{attribute 'no_explicit_call' := 'Do not call the body - Stick to OOP'}
(* XPlanar Environment - 1 per associated XPlanar 
	The Planar environment is a software object that represents the two-dimensional XPlanar stator surface. Together with Planar movers in a group, 
	it prevents collisions of the movers with the edge of the surface. *)
FUNCTION_BLOCK FB_XP_Environment EXTENDS FB_CH_Object IMPLEMENTS I_XP_Environment
VAR
	//Link to Planar-Environment object
	fbEnvironment : MC_PlanarEnvironment;
	fbUtilityEnvirement : FB_TcIoXPlanarEnvironment;
	
	{attribute 'hide'}  
	bInitDone :BOOL := FALSE;
	{attribute 'hide'}
	ipXpSystem : I_XP_System_Registration;
	{attribute 'hide'}               	
	fbFeedback 			: FB_XP_Feedback(ipSourceInfo := fbSourceInfo);	
	{attribute 'hide'}                   	
	eActiveCommand 		: CHALET_Nc.E_NcAxisCommands := CHALET_Nc.E_NcAxisCommands.None;
	{attribute 'hide'}
	bCollisionCheckEnabled : BOOL := TRUE;
	{attribute 'hide'}
	fMoverOffsetWarning : LREAL := 2.0; //[mm]
	{attribute 'hide'}
	fMoverOffsetError: LREAL := 0.0;//[mm]
	{attribute 'hide'}
	eMoverDetectionStatus : MoverDetectionStatus;
	{attribute 'hide'}
	eMoverDetectionStatusLastCycle : MoverDetectionStatus;
END_VAR


// Planar-Feedback objects
VAR
	{attribute 'hide'} 
	fbFeedbackAddToGrp : MC_PlanarFeedback;
	{attribute 'hide'} 
	fbFeedbackRmvFromGrp : MC_PlanarFeedback;
	{attribute 'hide'} 
	fbFeedbackConfigure : MC_PlanarFeedback;
	{attribute 'hide'} 
	fbFeedbackClear : MC_PlanarFeedback;
END_VAR

METHOD AddToGroup : HRESULT
VAR_INPUT
	iGroup : I_XP_Group;
END_VAR
IF NOT THIS^.fbFeedback.Busy THEN
	THIS^.eActiveCommand 				:= CHALET_NC.E_NcAxisCommands.AddToGroupe;
	THIS^.fbFeedback.ActiveCommand 		:= TO_STRING(THIS^.eActiveCommand);	
	THIS^.fbFeedback.LastCommandAccepted:= TRUE;		
	THIS^.fbFeedback.Busy 				:= TRUE;
	
	iGroup.AddEnvironment(THIS^.fbEnvironment, THIS^.fbFeedbackAddToGrp);
	AddToGroup := S_OK;
ELSE
	AddToGroup := S_FALSE;
	THIS^.fbFeedback.LastCommandAccepted:= FALSE;	
END_IF
END_METHOD

(* Clears the Planar Environment (stators and boundary). *)
METHOD Clear : HRESULT
THIS^.eActiveCommand 				:= CHALET_NC.E_NcAxisCommands.Clear;
THIS^.fbFeedback.ActiveCommand 		:= TO_STRING(THIS^.eActiveCommand);	
THIS^.fbFeedback.LastCommandAccepted:= TRUE;		
THIS^.fbFeedback.Busy 				:= TRUE;

THIS^.fbEnvironment.Clear(commandFeedback:=THIS^.fbFeedbackClear);
Clear := S_OK;
END_METHOD

{attribute 'monitoring':='call'}
(* If Enable, the movers are checked for collisions with each other.
Warning and error can have their own size offsets.
The error leads to a stop with higher dynamics.
In simulation, an error does not lead to a stop *)
PROPERTY CollisionCheck : BOOL
GET
CollisionCheck := THIS^.bCollisionCheckEnabled;
END_GET
SET
THIS^.bCollisionCheckEnabled := CollisionCheck;
END_SET
END_PROPERTY

//Return an interface to the mover if a collision is active else return 0. The check stops after the first collision found
METHOD PROTECTED CollisionDetectionAlgorithm : I_XP_Mover
VAR_INPUT
	ipListOfMovers : I_CH_LIST;
	fOffsetMoverSize : LREAL := 1.0; //Offset on the mover dimension from the MC3 mover object [mm];
END_VAR
VAR
	aPointsMover1 : ARRAY[0..3] OF  Tc3_Physics.PositionXY;
	aPointsEachMover : ARRAY[0..3] OF  Tc3_Physics.PositionXY;
	aPointsDelta : ARRAY[0..3] OF  Tc3_Physics.PositionXY;
	
	fMoverWidth, fMoverHight : LREAL;
	fMoverXPos, fMoverYPos, fMoverCPos : LREAL;
	
	ipMover1, ipEachMover : I_XP_Mover;
	fbListOfMoverToCheck : FB_CH_List;
	
	fAngle : LREAL;
	a, b, c: LREAL;
	Pa, Pb, Pc : REFERENCE TO Tc3_Physics.PositionXY;
	fcos : LREAL;
	
	nIdx, nIdxMover1, nIdxPlus1 : UINT;
	ipMover2CollisionFound : I_XP_Mover;
END_VAR
//Get all mover in a list
fbListOfMoverToCheck.Duplicate(ipListOfMovers);



//Check list for invalide Act Pos - ex.: if mover is not found 
fbListOfMoverToCheck.ResetIterator();
WHILE fbListOfMoverToCheck.HasNextObject() DO
	__QUERYINTERFACE(fbListOfMoverToCheck.GetNextObject(),ipMover1);
	
	IF ipMover1.MoverIsNotPresent THEN 		
		//remove from list
		fbListOfMoverToCheck.RemoveObject(ipMover1);
		
	END_IF
END_WHILE



fbListOfMoverToCheck.ResetIterator();
WHILE fbListOfMoverToCheck.HasNextObject() DO
	//get first mover in list,
	__QUERYINTERFACE(fbListOfMoverToCheck.GetNextObject(),ipMover1);
	
	fMoverXPos := ipMover1.PositionAct.x;
	fMoverYPos := ipMover1.PositionAct.y;
	fMoverCPos := ipMover1.PositionAct.c;
		
	//Get corner points of the rectangle 
	fMoverWidth := ipMover1.MoverWidth - fOffsetMoverSize;
	fMoverHight := ipMover1.MoverHeight - fOffsetMoverSize;
	aPointsMover1[0].SetValuesXY(x:= -fMoverWidth/2, y:= -fMoverHight/2);//Bottom Left
	aPointsMover1[1].SetValuesXY(x:= -fMoverWidth/2, y:=  fMoverHight/2);//Top Left
	aPointsMover1[2].SetValuesXY(x:=  fMoverWidth/2, y:=  fMoverHight/2);//Top Ritgh
	aPointsMover1[3].SetValuesXY(x:=  fMoverWidth/2, y:= -fMoverHight/2);//Bottom Rigth
	
	//Rotation of the mover
	F_RotatePositionXY(aPointsMover1[0], fMoverCPos);
	F_RotatePositionXY(aPointsMover1[1], fMoverCPos);
	F_RotatePositionXY(aPointsMover1[2], fMoverCPos);
	F_RotatePositionXY(aPointsMover1[3], fMoverCPos);
	
	//shift to mover coordinates
	aPointsMover1[0].ShiftByXY(dx:= fMoverXPos, dy:= fMoverYPos);
	aPointsMover1[1].ShiftByXY(dx:= fMoverXPos, dy:= fMoverYPos);
	aPointsMover1[2].ShiftByXY(dx:= fMoverXPos, dy:= fMoverYPos);
	aPointsMover1[3].ShiftByXY(dx:= fMoverXPos, dy:= fMoverYPos);
	
	
	//do an check for all mover
	fbListOfMoverToCheck.ResetIterator();
	WHILE fbListOfMoverToCheck.HasNextObject() DO
		__QUERYINTERFACE(fbListOfMoverToCheck.GetNextObject(),ipEachMover);
		
		//Skip if same
		IF ipEachMover = ipMover1 THEN
			CONTINUE;
		END_IF
		
		//Skip if far away
		IF (MAX(ipEachMover.MoverHeight, ipEachMover.MoverWidth) + MAX(ipMover1.MoverHeight, ipMover1.MoverWidth) + fOffsetMoverSize) < F_DistXYVectors(ipEachMover.PositionAct, ipMover1.PositionAct) THEN
			CONTINUE;
		END_IF
		
		
		fMoverXPos := ipEachMover.PositionAct.x;
		fMoverYPos := ipEachMover.PositionAct.y;
		fMovercPos := ipEachMover.PositionAct.c;
		
		//Get corner points of the rectangle 
		fMoverWidth := ipEachMover.MoverWidth - fOffsetMoverSize;
		fMoverHight := ipEachMover.MoverHeight - fOffsetMoverSize;
		aPointsEachMover[0].SetValuesXY(x:= -fMoverWidth/2, y:= -fMoverHight/2);//Bottom Left
		aPointsEachMover[1].SetValuesXY(x:= -fMoverWidth/2, y:=  fMoverHight/2);//Top Left
		aPointsEachMover[2].SetValuesXY(x:=  fMoverWidth/2, y:=  fMoverHight/2);//Top Ritgh
		aPointsEachMover[3].SetValuesXY(x:=  fMoverWidth/2, y:= -fMoverHight/2);//Bottom Rigth

		//Rotation of the mover
		F_RotatePositionXY(aPointsEachMover[0], fMoverCPos);
		F_RotatePositionXY(aPointsEachMover[1], fMoverCPos);
		F_RotatePositionXY(aPointsEachMover[2], fMoverCPos);
		F_RotatePositionXY(aPointsEachMover[3], fMoverCPos);
		
		//shift to mover coordinates
		aPointsEachMover[0].ShiftByXY(dx:= fMoverXPos, dy:= fMoverYPos);
		aPointsEachMover[1].ShiftByXY(dx:= fMoverXPos, dy:= fMoverYPos);
		aPointsEachMover[2].ShiftByXY(dx:= fMoverXPos, dy:= fMoverYPos);
		aPointsEachMover[3].ShiftByXY(dx:= fMoverXPos, dy:= fMoverYPos);		
		
		//check each corener if inside each mover
		FOR nIdxMover1 := 0 TO 3 DO
			
			(* A triangle is created between a corner point of Mover1 (point a) and two corner points of Mover2 (points B and C). 
			All corner points of Mover2 are now tested one after the other. If the sum of all angles "a" is 360 degrees, 
			then point A is inside mover 2 and there is a collision *)
			fAngle := 0;
			FOR nIdx := 0 TO 3 DO
				nIdxPlus1 := ((nIdx+1)MOD 4);
			
				Pa REF= aPointsMover1[nIdxMover1];
				Pb REF= aPointsEachMover[nIdx];
				Pc REF= aPointsEachMover[nIdxPlus1];					
				

				a := SQRT(EXPT((Pb.x - Pc.x),2)+EXPT((Pb.y - Pc.y),2));
				b := SQRT(EXPT((Pa.x - Pc.x),2)+EXPT((Pa.y - Pc.y),2));
				c := SQRT(EXPT((Pa.x - Pb.x),2)+EXPT((Pa.y - Pb.y),2));
				
				
				IF b=0 OR c=0 THEN
					//Error - Return the found mover
					CollisionDetectionAlgorithm := ipMover1;
					//with which mover is the collision
					ipMover2CollisionFound := ipEachMover;
					RETURN;
				ELSE
					(*  a/sin(α) = b/sin(β) = c/sin(γ) *)
					fcos := (EXPT(b,2) + EXPT(c,2) - EXPT(a,2))/(2*b*c);
					fcos := LIMIT(-1.0, fcos, 1.0);
					fAngle :=  fAngle + ACOS(fcos);
				END_IF
			END_FOR
			
			//if the point is inside the mover, the sum of all angles is exactly 360°-> 2pi
			IF ABS(fAngle - 2*Tc2_System.PI)<0.01 THEN
				//Error - Return the found mover
				CollisionDetectionAlgorithm := ipMover1;
				//with which mover is the collision
				ipMover2CollisionFound := ipEachMover;
				RETURN;
			END_IF
			
		END_FOR

	END_WHILE
	fbListOfMoverToCheck.RestoreIterator();
	
	
	
END_WHILE
END_METHOD

METHOD Configure : HRESULT
THIS^.eActiveCommand 				:= CHALET_NC.E_NcAxisCommands.Configure;
THIS^.fbFeedback.ActiveCommand 		:= TO_STRING(THIS^.eActiveCommand);	
THIS^.fbFeedback.LastCommandAccepted:= TRUE;		
THIS^.fbFeedback.Busy 				:= TRUE;

THIS^.fbEnvironment.CreateBoundary(commandFeedback:=THIS^.fbFeedbackConfigure);
Configure := S_OK;
END_METHOD

METHOD FB_init : BOOL
VAR_INPUT
	bInitRetains : BOOL; // if TRUE, the retain variables are initialized (warm start / cold start)
	bInCopyCode : BOOL;  // if TRUE, the instance afterwards gets moved into the copy code (online change)
	
	ipSystem : I_CH_Object;
END_VAR
//Do the following code once during start up and not during onlinechange
IF NOT bInCopyCode THEN 
	
	(* Register to the Xplanar System
	   1. Test if the interface exists
	   2. Test if the object implements a "System for Mover" interface 
	*)
	IF ipSystem <> 0 AND_THEN __QUERYINTERFACE(ipSystem,THIS^.ipXpSystem) THEN
		THIS^.ipXpSystem.LinkEnvironment(THIS^);
	END_IF
	
	
	THIS^.fbFeedback.ActiveCommand 		:= TO_STRING(THIS^.eActiveCommand);	
	
END_IF
END_METHOD

{attribute 'monitoring':='call'}
PROPERTY Feedback : I_XP_Feedback
GET
Feedback := THIS^.fbFeedback;
END_GET
END_PROPERTY

METHOD Initialize : HRESULT
VAR
	stVarInfo : __SYSTEM.VAR_INFO;
END_VAR
VAR_INST
	//This error cannot be reset. Requires a reset cold
	{attribute 'hide'}	
	fbInitError : FB_TcAlarm;
END_VAR
// Check if link to envirement is mapped
IF NOT THIS^.Mapped THEN
	IF NOT fbInitError.bRaised THEN 
		//This error cannot be reset. Requires a reset cold
		fbInitError.CreateEx(stEventEntry:=TC_EVENTS.CHALET_Base_Events.VariableLinkMissing, ipSourceInfo := THIS^.fbSourceInfo, bWithConfirmation := FALSE);
		stVarInfo := __VARINFO(fbEnvironment);
		fbInitError.ipArguments.AddString(stVarInfo.Symbol);
		fbInitError.Raise(0);
	END_IF
	Initialize := E_FAIL;
	RETURN;
END_IF



IF NOT bInitDone THEN
	//Busy
	Initialize := S_PENDING;
	
	IF fbUtilityEnvirement.Init(bExecute := TRUE) THEN
		fbUtilityEnvirement.Init(bExecute := FALSE);
		bInitDone := TRUE;
	END_IF
	
	
ELSE	
	//Done
	Initialize := S_OK;
END_IF


THIS^.eActiveCommand 				:= CHALET_NC.E_NcAxisCommands.Initialize;
THIS^.fbFeedback.ActiveCommand 		:= TO_STRING(THIS^.eActiveCommand);	
THIS^.fbFeedback.LastCommandAccepted:= TRUE;	
//Set done or keep in busy state	
THIS^.fbFeedback.HR := Initialize;
END_METHOD

{attribute 'monitoring':='call'}
PROPERTY Mapped : BOOL //Project is mapped to MC (McToPlc and PlcToMc)
GET
VAR
	bMcToPlcNotMapped 	: BOOL;
END_VAR
bMcToPlcNotMapped := F_GetMappingStatus(ADR(THIS^.fbEnvironment.MCTOPLC_STD), SIZEOF(THIS^.fbEnvironment.MCTOPLC_STD)) <> EPlcMappingStatus.MS_Mapped;

Mapped := NOT bMcToPlcNotMapped;
END_GET
END_PROPERTY

{attribute 'monitoring':='call'}
//Offset on the mover dimension from the MC3 mover object [mm] ;
// >0 menas the warning is earlier
PROPERTY MoverCollisionOffsetError : LREAL
GET
MoverCollisionOffsetError := fMoverOffsetError;
END_GET
SET
fMoverOffsetError := MoverCollisionOffsetError;
END_SET
END_PROPERTY

{attribute 'monitoring':='call'}
//Offset on the mover dimension from the MC3 mover object [mm] ;
// >0 menas the warning is earlier
PROPERTY MoverCollisionOffsetWarning : LREAL
GET
MoverCollisionOffsetWarning :=  fMoverOffsetWarning;
END_GET
SET
fMoverOffsetWarning := MoverCollisionOffsetWarning;
END_SET
END_PROPERTY

{attribute 'monitoring':='call'}
//Unique object ID
PROPERTY OID : OTCID
GET
OID := THIS^.fbEnvironment.MCTOPLC_STD.EnvironmentOID;
END_GET
END_PROPERTY

{attribute 'monitoring':='call'}
PROPERTY PlanarEnvironment : REFERENCE TO MC_PlanarEnvironment
GET
PlanarEnvironment ref= THIS^.fbEnvironment;
END_GET
END_PROPERTY

(* Time-critical information is processed here, which can then be polled via the property every cycle. 
The update method is usually at the end of the program and then it is already 'outdated'. *)
METHOD PRIVATE Prepare : HRESULT
VAR CONSTANT
	N_IDX_OFFSET_MoverDetectionStatus 	: UDINT := 16#03171005; // Parameter(online) in Planar  Processing Unit object 
END_VAR
VAR
	nParaSize : UDINT;
	pParaData : PVOID;
	hr : HRESULT;
	ipComObject : ITComObject;
END_VAR
VAR_INST
	{attribute 'hide'}
	nLastUpdatedCycleCount : UDINT;
END_VAR
//Check if this Cycle the dates are allready prepared
IF nLastUpdatedCycleCount <> TwinCAT_SystemInfoVarList._TaskInfo[THIS^.nTaskIndex].CycleCount THEN
	nLastUpdatedCycleCount := TwinCAT_SystemInfoVarList._TaskInfo[THIS^.nTaskIndex].CycleCount;

	
	//************** Read MoverDetectionStatus **************
	//Get interface to ComObject
	FW_ObjMgr_GetObjectInstance(oid:= THIS^.ProcessingUnitOID, iid:= TC_GLOBAL_IID_LIST.IID_ITComObject, pipUnk:= ADR(ipComObject));
	
	//Get ADR and SIZE
	nParaSize := SIZEOF(eMoverDetectionStatus);	pParaData := ADR(eMoverDetectionStatus);
	
	IF ipComObject <> 0 THEN
		hr := ipComObject.TcGetObjPara(pid:=N_IDX_OFFSET_MoverDetectionStatus , nData:= nParaSize, pData:= pParaData, pgp:=0 );	
		FW_SafeRelease(ADR(ipComObject));
	END_IF
	
	//force to have the in progress active FOR 1 cycle longer
	IF eMoverDetectionStatus = MoverDetectionStatus.DetectionSuccessful AND eMoverDetectionStatusLastCycle = MoverDetectionStatus.DetectionInProcess THEN
		//Store info from last cycle
		eMoverDetectionStatusLastCycle := eMoverDetectionStatus;
		eMoverDetectionStatus := MoverDetectionStatus.DetectionInProcess;
	ELSE	
		//Store info from last cycle
		eMoverDetectionStatusLastCycle := eMoverDetectionStatus;
	END_IF
	


		
END_IF
END_METHOD

{attribute 'monitoring':='call'}
//Enumeration MoverDetectionStatus
PROPERTY ProcessingUnitMoverDetectionStatus : MoverDetectionStatus
GET
THIS^.Prepare();//Prepare time-critical information, if not already done


ProcessingUnitMoverDetectionStatus := THIS^.eMoverDetectionStatus;
END_GET
END_PROPERTY

{attribute 'monitoring':='call'}
//Object ID of the IoXPlanar processing unit
PROPERTY ProcessingUnitOID : OTCID
GET
VAR
	nProcessingUnitOid : OTCID;
END_VAR
VAR CONSTANT
	N_IDX_OFFSET_PU_Oid 	: UDINT := 16#050300C0; // Parameter(online) in Planar Environment object 
END_VAR

VAR
	nParaSize : UDINT;
	pParaData : PVOID;
	hr : HRESULT;
	ipComObject : ITComObject;
	nOid : OTCID;
END_VAR
//Get TcCom Object ID
nOid := THIS^.OID;

//Get interface to ComObject
FW_ObjMgr_GetObjectInstance(oid:= nOid, iid:= TC_GLOBAL_IID_LIST.IID_ITComObject, pipUnk:= ADR(ipComObject));

//Get ADR and SIZE
nParaSize := SIZEOF(nProcessingUnitOid);	pParaData := ADR(nProcessingUnitOid);

IF ipComObject <> 0 THEN
	hr := ipComObject.TcGetObjPara(pid:=N_IDX_OFFSET_PU_Oid , nData:= nParaSize, pData:= pParaData, pgp:=0 );	
	FW_SafeRelease(ADR(ipComObject));
END_IF

ProcessingUnitOID := nProcessingUnitOid;
END_GET
END_PROPERTY

METHOD RemoveFromGroup : HRESULT
IF NOT THIS^.fbFeedback.Busy THEN
	THIS^.eActiveCommand 				:= CHALET_NC.E_NcAxisCommands.RemoveFromGroupe;
	THIS^.fbFeedback.ActiveCommand 		:= TO_STRING(THIS^.eActiveCommand);	
	THIS^.fbFeedback.LastCommandAccepted:= TRUE;		
	THIS^.fbFeedback.Busy 				:= TRUE;
	
	THIS^.fbEnvironment.RemoveFromGroup(THIS^.fbFeedbackRmvFromGrp);
	RemoveFromGroup := S_OK;
ELSE
	RemoveFromGroup := S_FALSE;
	THIS^.fbFeedback.LastCommandAccepted:= FALSE;	
END_IF
END_METHOD

{attribute 'monitoring':='call'}
//Interface to CHALET system to which this object belongs
PROPERTY System : I_XP_System_PLC
GET
//get I_x_System_PLC interface from I_x_System_Registration
__QUERYINTERFACE(THIS^.ipXpSystem, System);
END_GET
END_PROPERTY

METHOD PUBLIC Update : HRESULT



// ********************** Set feedback depending on active command *******************************
CASE THIS^.eActiveCommand OF
	E_NcAxisCommands.None: 
		//Display if a Mover Error is active during no command is active
		IF THIS^.fbEnvironment.Error AND NOT fbFeedback.Error THEN 
			fbFeedback.ErrorId 			:= THIS^.fbEnvironment.ErrorID;
			fbFeedback.ActiveCommand 	:= TO_STRING(E_NcAxisCommands.None);	
			fbFeedback.ClearObjectInfo();
		END_IF

	E_NcAxisCommands.Initialize:
		fbFeedback.Busy 			:= NOT THIS^.bInitDone;
		fbFeedback.Done 			:= THIS^.bInitDone;
		fbFeedback.ErrorId 			:= 0;
		fbFeedback.ClearObjectInfo();
		                                                       			                        	
	E_NcAxisCommands.Clear:     	
		fbFeedback.Busy 			:= fbFeedbackClear.Busy;
		fbFeedback.Done 			:= fbFeedbackClear.Done;
		fbFeedback.ErrorId 			:= fbFeedbackClear.ErrorID;
        fbFeedback.ObjectInfo		:= fbFeedbackClear.objectInfo;
           			                        	
	E_NcAxisCommands.Configure:     	
		fbFeedback.Busy 			:= fbFeedbackConfigure.Busy;
		fbFeedback.Done 			:= fbFeedbackConfigure.Done;
		fbFeedback.ErrorId 			:= fbFeedbackConfigure.ErrorID;
        fbFeedback.ObjectInfo		:= fbFeedbackConfigure.objectInfo;
                                      			                        	
	E_NcAxisCommands.AddToGroupe:     	
		fbFeedback.Busy 			:= fbFeedbackAddToGrp.Busy;
		fbFeedback.Done 			:= fbFeedbackAddToGrp.Done;
		fbFeedback.ErrorId 			:= fbFeedbackAddToGrp.ErrorID;
        fbFeedback.ObjectInfo		:= fbFeedbackAddToGrp.objectInfo;
                                      			                        	
	E_NcAxisCommands.RemoveFromGroupe:     	
		fbFeedback.Busy 			:= fbFeedbackRmvFromGrp.Busy;
		fbFeedback.Done 			:= fbFeedbackRmvFromGrp.Done;
		fbFeedback.ErrorId 			:= fbFeedbackRmvFromGrp.ErrorID;
        fbFeedback.ObjectInfo		:= fbFeedbackRmvFromGrp.objectInfo;
                                		
	ELSE//External command in subclass
		;
END_CASE


// **********************  Stop to execute commands on .done or .error ***************************
IF fbFeedback.Done OR THIS^.fbFeedback.Error THEN
	eActiveCommand 				:= E_NcAxisCommands.None;
END_IF





//Update Collision subroutin
THIS^.UpdateCollisionDetection();


//Update xplanar object
THIS^.fbEnvironment.Update();

//Update feedback object
fbFeedbackConfigure.Update(); 
fbFeedbackClear.Update(); 
fbFeedbackAddToGrp.Update(); 
fbFeedbackRmvFromGrp.Update();
END_METHOD

METHOD PROTECTED UpdateCollisionDetection : HRESULT
VAR
	bDisableDuringMoverDetection : BOOL;
	ipMoverCollision : I_XP_Mover;
	ipSystemPlc : I_XP_System_PLC;
	nX, nY : DINT;
END_VAR
VAR_INST
	{attribute 'hide'}	
	ipMoverCollisionOldWarning : I_XP_Mover;
	{attribute 'hide'}	
	fbAlarmCollisionMoverWarning : FB_TcAlarm;	
	{attribute 'hide'}	
	ipMoverCollisionOldAlarm : I_XP_Mover;
	{attribute 'hide'}	
	fbAlarmCollisionMoverAlarm : FB_TcAlarm;
END_VAR
bDisableDuringMoverDetection := THIS^.ProcessingUnitMoverDetectionStatus = MoverDetectionStatus.DetectionInProcess;


//Check whether a mover has a collision with another mover and generate a warning.
//Only 1 mover is found and displayed
//WARNING - each mover default is 2mm larger
IF THIS^.bCollisionCheckEnabled AND NOT bDisableDuringMoverDetection THEN
	//get mover or 0 for no collision
	ipMoverCollision := CollisionDetectionAlgorithm(fOffsetMoverSize := THIS^.fMoverOffsetWarning, ipListOfMovers := THIS^.ipXpSystem.MoversPresent);
	
	IF ipMoverCollision <> 0 AND_THEN ipMoverCollision <> ipMoverCollisionOldWarning AND_THEN NOT ipMoverCollision.MoverIsNotPresent THEN
		fbAlarmCollisionMoverWarning.CreateEx(tc_Events.CHALET_XPlanar_Events.MoverCollisionWarning, 0, THIS^.fbSourceInfo);
		//Mover "{0}" has a collision with another mover at position X:{1} Y:{2}
		nX := LREAL_TO_DINT(ipMoverCollision.PlanarMover.MCTOPLC.ACT.ActPos.x);
		nY := LREAL_TO_DINT(ipMoverCollision.PlanarMover.MCTOPLC.ACT.ActPos.y);
		fbAlarmCollisionMoverWarning.ipArguments.Clear().AddStringByValue(ipMoverCollision.LUID).AddDInt(nX).AddDint(nY);
		fbAlarmCollisionMoverWarning.Raise(0);
	ELSIF ipMoverCollision = 0 THEN
		//No collision found
		fbAlarmCollisionMoverWarning.Clear(0,0);
	END_IF
	ipMoverCollisionOldWarning := ipMoverCollision;
ELSE
	fbAlarmCollisionMoverWarning.Clear(0,0);
	ipMoverCollisionOldWarning := 0;
END_IF

//Check whether a mover has a collision with another mover and generate a warning.
//Only 1 mover is found and displayed
//ERROR - each mover is default -1mm smaller
IF THIS^.bCollisionCheckEnabled AND NOT bDisableDuringMoverDetection  THEN
	//get mover or 0 for no collision
	ipMoverCollision := CollisionDetectionAlgorithm(fOffsetMoverSize := THIS^.fMoverOffsetError, ipListOfMovers := THIS^.ipXpSystem.MoversPresent);
	
	IF ipMoverCollision <> 0 AND ipMoverCollision <> ipMoverCollisionOldAlarm THEN
		fbAlarmCollisionMoverAlarm.CreateEx(tc_Events.CHALET_XPlanar_Events.MoverCollisionStop, 0, THIS^.fbSourceInfo);
		//Mover "{0}" has a collision with another mover at position X:{1} Y:{2}
		fbAlarmCollisionMoverAlarm.ipArguments.AddStringByValue(ipMoverCollision.LUID).AddUDInt(LREAL_TO_UDINT(ipMoverCollision.PlanarMover.MCTOPLC.ACT.ActPos.x)).AddUDInt(LREAL_TO_UDINT(ipMoverCollision.PlanarMover.MCTOPLC.ACT.ActPos.y));
		fbAlarmCollisionMoverAlarm.Raise(0);

		//Stop if this is a real system, keep running in simulation
		
		IF THIS^.UtilityEnvirement.TcIoXpu(1).GetOperationMode() = XplanarOperationMode.Normal THEN
			IF __QUERYINTERFACE(THIS^.ipXpSystem, ipSystemPlc) THEN
				//Disable System
				ipSystemPlc.FastStop();
			END_IF
		END_IF
	ELSIF ipMoverCollision = 0 THEN
		//No collision found
		fbAlarmCollisionMoverAlarm.Clear(0,0);
	END_IF
		
	ipMoverCollisionOldAlarm := ipMoverCollision;
ELSE
	fbAlarmCollisionMoverAlarm.Clear(0,0);
	ipMoverCollisionOldAlarm := 0;
END_IF
END_METHOD

{attribute 'monitoring':='call'}
PROPERTY UtilityEnvirement : Tc3_XPlanarUtility.I_Environment
GET
UtilityEnvirement := fbUtilityEnvirement;
END_GET
END_PROPERTY

END_FUNCTION_BLOCK

(* stored: Version 1.1.0.1, ProductVersion 3.1.4024.15
   POU FB_XP_Environment: Id {6c9df844-5691-4d75-a14e-01fa98bb26e3}, SpecialFunc None
   Folder CollisionDetection: Id {cc9e35ec-135a-40d8-8e41-0acd41982d0a}
   Folder Group: Id {1ec64b27-6c0b-4188-9c58-0a330b77e507}
   Method AddToGroup: Id {287f1c1d-9530-419a-a6a6-4458e419ac5b}
   Method Clear: Id {e2df5771-2b46-447a-a790-27cc8fd54fd0}
   Property CollisionCheck: Id {5d152728-5cec-4b17-9311-3f3e2bf04bf5}
   Get Get: Id {54935009-1b45-4fd3-9061-4a30085d2687}
   Set Set: Id {00ab7b05-80a1-4d9a-912d-ef7d9e157a78}
   Method CollisionDetectionAlgorithm: Id {aeea7fd2-2f60-42db-8d11-f0607822de9c}
   Method Configure: Id {94a277cb-a6e6-4475-a159-23a2d173207d}
   Method FB_init: Id {3332ee11-a20c-443f-8062-eeaf7c0acaa7}
   Property Feedback: Id {4d454920-2471-4339-ada8-e58505a82219}
   Get Get: Id {92adf6cc-8743-45e1-869d-653b09b7978d}
   Method Initialize: Id {40324653-7238-423b-a8fd-05ed7a18c09e}
   Property Mapped: Id {b8d25027-a67e-470b-9581-b959c6328df3}
   Get Get: Id {bb7d8e37-da00-480b-964e-962762127f9f}
   Property MoverCollisionOffsetError: Id {de9a372c-f660-48c5-b2b6-268474f6d44b}
   Get Get: Id {ade65951-3360-4b37-9211-03998904bcf1}
   Set Set: Id {b2fc7742-cf8c-451a-97a8-ec1b9fa15b0d}
   Property MoverCollisionOffsetWarning: Id {2640c673-abce-4176-be6e-b2167e877f28}
   Get Get: Id {6b38c531-fcff-44b0-934f-a666556d7281}
   Set Set: Id {88baf0ce-9d1b-476a-8a5f-ee5a5f8b4018}
   Property OID: Id {7ae2b0fe-be79-4b9e-9fc2-a7d176f204c5}
   Get Get: Id {88f94db8-1661-4f49-b868-d54d29985f73}
   Property PlanarEnvironment: Id {a6c655b1-a79b-420b-8a88-eca38ef9d746}
   Get Get: Id {26cfa0c3-4ea1-4baa-9ed5-8f88fba409a0}
   Method Prepare: Id {14ed7006-68ff-4b31-ab84-f5289abed286}
   Property ProcessingUnitMoverDetectionStatus: Id {e2cf85a4-d4a6-4c0e-84f4-a50580e7f0f4}
   Get Get: Id {6fc52da6-863a-4af1-85a2-8b9ff7f7a3d3}
   Property ProcessingUnitOID: Id {755616fb-b190-4a32-9b97-8c58500630c9}
   Get Get: Id {da73534b-1724-4d81-8aca-f6998aa8fb37}
   Method RemoveFromGroup: Id {b08ba9a4-1133-4063-9835-12556583929a}
   Property System: Id {39ffeb45-ee5e-4724-be7c-c11cc9e33b10}
   Get Get: Id {ec0f323d-84f2-44b2-afcb-d65582a62b18}
   Method Update: Id {476a95ad-3269-45e6-a01b-247748d45f7c}
   Method UpdateCollisionDetection: Id {a9513029-f962-44c5-9b2b-a1a01d10798b}
   Property UtilityEnvirement: Id {2e740e9d-ce68-40bf-aad7-1f44d441a8bc}
   Get Get: Id {722af0ec-c8ab-4b67-b67b-63ac0647ba49} *)
